(* PLC project Tc2_Utilities.CONCAT2 Demo, tc3-libraries-kb TwinCAT 3.1 *)
(* stored: creationDateTime 2026-05-10T16:00:00, modificationDateTime 2026-05-10T16:00:00 *)

PROGRAM P_Demo_CONCAT2
  VAR
    rResult : BOOL;  (* CONCAT2 返回值 *)
    bRun : BOOL;  (* 触发一次调用 *)
    sA : STRING;  (* 测试用本地变量 *)
    sB : STRING;  (* 测试用本地变量 *)
    sC : STRING;  (* 测试用本地变量 *)
  END_VAR

            // ============================================================
// Tc2_Utilities.CONCAT2 演示程序（FUNCTION）
// ============================================================
// 验证步骤：
//   1. 引用 Tc2_Utilities
//   2. 编译 + 登录
//   3. 强制 bRun := TRUE 一个周期
//   4. 在线监视 rResult / 各 demo 变量
// ============================================================

sA := 'Hello, '; sB := 'World!';
IF bRun THEN
    rResult := CONCAT2(ADR(sA), ADR(sB), ADR(sC), SIZEOF(sC));
    bRun := FALSE;
END_IF;

          
END_PROGRAM
